// TIA Portal V20 export
VAR_GLOBAL   // PLC tag table "Unit1Em8"
   "BA060ZSIBK14.00" AT %I1052.0 : Bool;   // (HOME) HIPOT TAB CONTACTOR BACKWARD
   "BA060ZSIBK14.01" AT %I1052.1 : Bool;   // (HOME) HIPOT TAB CONTACTOR LEFT OPEN
   "BA060ZSIBK14.02" AT %I1052.2 : Bool;   // (HOME) HIPOT TAB CONTACTOR RIGHT OPEN
   "BA060ZSIBK14.03" AT %I1052.3 : Bool;   // SPARE
   "BA060ZSIBK14.04" AT %I1052.4 : Bool;   // SPARE
   "BA060ZSIBK14.05" AT %I1052.5 : Bool;   // (HOME) INSPECTION (HIPOT&THICKNESS) STAGE LIFT FRONT DOWN
   "BA060ZSIBK14.06" AT %I1052.6 : Bool;   // (HOME) INSPECTION (HIPOT&THICKNESS) STAGE LIFT REAR DOWN
   "BA060ZSIBK14.07" AT %I1052.7 : Bool;   // SPARE
   "BA060ZSIBK14.08" AT %I1053.0 : Bool;   // (WORK) HIPOT TAB CONTACTOR FORWARD
   "BA060ZSIBK14.09" AT %I1053.1 : Bool;   // (WORK) HIPOT TAB CONTACTOR LEFT CLOSE
   "BA060ZSIBK14.10" AT %I1053.2 : Bool;   // (WORK) HIPOT TAB CONTACTOR RIGHT CLOSE
   "BA060ZSIBK14.11" AT %I1053.3 : Bool;   // SPARE
   "BA060ZSIBK14.12" AT %I1053.4 : Bool;   // SPARE
   "BA060ZSIBK14.13" AT %I1053.5 : Bool;   // (WORK) INSPECTION (HIPOT&THICKNESS) STAGE LIFT FRONT UP
   "BA060ZSIBK14.14" AT %I1053.6 : Bool;   // (WORK) INSPECTION (HIPOT&THICKNESS) STAGE LIFT REAR UP
   "BA060ZSIBK14.15" AT %I1053.7 : Bool;   // SPARE
   "BA060ZSIBK15.02" AT %I1056.2 : Bool;   // HIPOT&THICKNESS STACK DETECT SENSOR
   "BA060ZSIBK15.03" AT %I1056.3 : Bool;   // HI-POT SAFETY PIN LOADING SENSOR
   "BA060ZSIBK15.04" AT %I1056.4 : Bool;   // SPARE
   "BA060ZSIBK15.05" AT %I1056.5 : Bool;   // SPARE
   "BA060ZSIBK15.06" AT %I1056.6 : Bool;   // SPARE
   "BA060ZSIBK15.07" AT %I1056.7 : Bool;   // SPARE
   "BA060ZSIBK15.09" AT %I1057.1 : Bool;   // SPARE
   "BA060ZSIBK15.10" AT %I1057.2 : Bool;   // SPARE
   "BA060ZSIBK15.11" AT %I1057.3 : Bool;   // SPARE
   "BA060ZSIBK15.12" AT %I1057.4 : Bool;   // SPARE
   "BA060ZSIBK15.13" AT %I1057.5 : Bool;   // SPARE
   "BA060ZSIBK15.14" AT %I1057.6 : Bool;   // SPARE
   "BA060ZSIBK15.15" AT %I1057.7 : Bool;   // SPARE
   "BA060AZSISP501.10" AT %I3001.0 : Bool;   // SPARE
   "BA060AZSISP501.11" AT %I3001.1 : Bool;   // SPARE
   "BA060AZSISP501.12" AT %I3001.2 : Bool;   // SPARE
   "BA060AZSISP501.13" AT %I3001.3 : Bool;   // SPARE
   "BA060AZSISP501.14" AT %I3001.4 : Bool;   // SPARE
   "BA060AZSISP501.15" AT %I3001.5 : Bool;   // SPARE
   "BA060AZSISP501.16" AT %I3001.6 : Bool;   // SPARE
   "BA060AZSISP501.17" AT %I3001.7 : Bool;   // SPARE
   "BA060ZSIPM08.00" AT %Q2028.0 : Bool;   // (WORK) HIPOT TAB CONTACTOR FORWARD
   "BA060ZSIPM08.01" AT %Q2028.1 : Bool;   // (HOME) HIPOT TAB CONTACTOR BACKWARD
   "BA060ZSIPM08.02" AT %Q2028.2 : Bool;   // (WORK) HIPOT TAB CONTACTOR LEFT CLOSE
   "BA060ZSIPM08.03" AT %Q2028.3 : Bool;   // (HOME) HIPOT TAB CONTACTOR LEFT OPEN
   "BA060ZSIPM08.04" AT %Q2028.4 : Bool;   // (WORK) HIPOT TAB CONTACTOR RIGHT CLOSE
   "BA060ZSIPM08.05" AT %Q2028.5 : Bool;   // (HOME) HIPOT TAB CONTACTOR RIGHT OPEN
   "BA060ZSIPM08.06" AT %Q2028.6 : Bool;   // SPARE
   "BA060ZSIPM08.07" AT %Q2028.7 : Bool;   // SPARE
   "BA060ZSIPM08.10" AT %Q2029.0 : Bool;   // SPARE
   "BA060ZSIPM08.11" AT %Q2029.1 : Bool;   // SPARE
   "BA060ZSIPM08.12" AT %Q2029.2 : Bool;   // (WORK) HIPOT & THICKNESS STAGE LIFT FRONT UP
   "BA060ZSIPM08.13" AT %Q2029.3 : Bool;   // (HOME) HIPOT & THICKNESS STAGE LIFT FRONT DOWN
   "BA060ZSIPM08.14" AT %Q2029.4 : Bool;   // (WORK) HIPOT & THICKNESS STAGE LIFT REAR DOWN
   "BA060ZSIPM08.15" AT %Q2029.5 : Bool;   // (HOME) HIPOT & THICKNESS STAGE LIFT REAR UP
   "BA060ZSIPM08.16" AT %Q2029.6 : Bool;   // SPARE
   "BA060ZSIPM08.17" AT %Q2029.7 : Bool;   // SPARE
   "BA060AZSISP504.10" AT %Q3001.0 : Bool;   // SPARE
   "BA060AZSISP504.11" AT %Q3001.1 : Bool;   // SPARE
   "BA060AZSISP504.12" AT %Q3001.2 : Bool;   // SPARE
   "BA060AZSISP504.13" AT %Q3001.3 : Bool;   // SPARE
   "BA060AZSISP504.14" AT %Q3001.4 : Bool;   // SPARE
   "BA060AZSISP504.15" AT %Q3001.5 : Bool;   // SPARE
   "BA060AZSISP504.16" AT %Q3001.6 : Bool;   // SPARE
   "BA060AZSISP504.17" AT %Q3001.7 : Bool;   // SPARE
END_VAR
VAR_GLOBAL CONSTANT   // user constants
   U1EM8_JOB01 : DInt := 1;   // ID for Job1
   U1EM8_JOB02 : DInt := 2;   // ID for Job2
   U1EM8_JOB03 : DInt := 3;   // ID for Job3
   U1EM8_JOB04 : DInt := 4;   // ID for Job4
   U1EM8_JOB05 : DInt := 5;   // ID for Job5
   U1EM8_JOB06 : DInt := 6;   // Starts with 1. E.g., the value means that axes exist.
   U1EM8_JOB07 : DInt := 7;
   U1EM8_JOB08 : DInt := 8;
   U1EM8_JOB09 : DInt := 9;
   U1EM8_JOB10 : DInt := 10;
   U1EM8_JOB11 : DInt := 11;
   U1EM8_JOB12 : DInt := 12;
   U1EM8_JOB13 : DInt := 13;
   U1EM8_JOB14 : DInt := 14;
   U1EM8_JOB15 : DInt := 15;
   U1EM8_JOB16 : DInt := 16;
   U1EM8_JOB17 : DInt := 17;
   U1EM8_JOB18 : DInt := 18;
   U1EM8_JOB19 : DInt := 19;
   U1EM8_JOB20 : DInt := 20;
   U1EM8_JOB21 : DInt := 21;
   U1EM8_JOB22 : DInt := 22;
   U1EM8_JOB23 : DInt := 23;
   U1EM8_JOB24 : DInt := 24;
   U1EM8_JOB25 : DInt := 25;
   U1EM8_JOB26 : DInt := 26;
   U1EM8_JOB27 : DInt := 27;
   U1EM8_JOB28 : DInt := 28;
   U1EM8_JOB29 : DInt := 29;
   U1EM8_JOB30 : DInt := 30;
   U1EM8_JOB31 : DInt := 31;
   U1EM8_JOB32 : DInt := 32;
   U1EM8_JOB33 : DInt := 33;
   U1EM8_JOB34 : DInt := 34;
   U1EM8_JOB35 : DInt := 35;
   U1EM8_JOB36 : DInt := 36;
   U1EM8_JOB37 : DInt := 37;
   U1EM8_JOB38 : DInt := 38;
   U1EM8_JOB39 : DInt := 39;
   U1EM8_JOB40 : DInt := 40;
   U1EM8_JOB41 : DInt := 41;
   U1EM8_JOB42 : DInt := 42;
   U1EM8_JOB43 : DInt := 43;
   U1EM8_JOB44 : DInt := 44;
   U1EM8_JOB45 : DInt := 45;
   U1EM8_JOB46 : DInt := 46;
   U1EM8_JOB47 : DInt := 47;
   U1EM8_JOB48 : DInt := 48;
   U1EM8_JOB49 : DInt := 49;
   U1EM8_JOB50 : DInt := 50;
   U1EM8_JOB51 : DInt := 51;
   U1EM8_JOB52 : DInt := 52;
   U1EM8_JOB53 : DInt := 53;
   U1EM8_JOB54 : DInt := 54;
   U1EM8_JOB55 : DInt := 55;
   U1EM8_JOB56 : DInt := 56;
   U1EM8_JOB57 : DInt := 57;
   U1EM8_JOB58 : DInt := 58;
   U1EM8_JOB59 : DInt := 59;
   U1EM8_JOB60 : DInt := 60;
   U1EM8_JOB61 : DInt := 61;
   U1EM8_JOB62 : DInt := 62;
   U1EM8_JOB63 : DInt := 63;
   U1EM8_JOB64 : DInt := 64;
   U1EM8_JOB65 : DInt := 65;
   U1EM8_JOB66 : DInt := 66;
   U1EM8_JOB67 : DInt := 67;
   U1EM8_JOB68 : DInt := 68;
   U1EM8_JOB69 : DInt := 69;
   U1EM8_JOB70 : DInt := 70;
   U1EM8_JOB71 : DInt := 71;
   U1EM8_JOB72 : DInt := 72;
   U1EM8_JOB73 : DInt := 73;
   U1EM8_JOB74 : DInt := 74;
   U1EM8_JOB75 : DInt := 75;
   U1EM8_JOB76 : DInt := 76;
   U1EM8_JOB77 : DInt := 77;
   U1EM8_JOB78 : DInt := 78;
   U1EM8_JOB79 : DInt := 79;
   U1EM8_JOB80 : DInt := 80;
   U1EM8_JOB81 : DInt := 81;
   U1EM8_JOB82 : DInt := 82;
   U1EM8_JOB83 : DInt := 83;
   U1EM8_JOB84 : DInt := 84;
   U1EM8_JOB85 : DInt := 85;
   U1EM8_JOB86 : DInt := 86;
   U1EM8_JOB87 : DInt := 87;
   U1EM8_JOB88 : DInt := 88;
   U1EM8_JOB89 : DInt := 89;
   U1EM8_JOB90 : DInt := 90;
   U1EM8_JOB91 : DInt := 91;
   U1EM8_JOB92 : DInt := 92;
   U1EM8_JOB93 : DInt := 93;
   U1EM8_JOB94 : DInt := 94;
   U1EM8_JOB95 : DInt := 95;
   U1EM8_JOB96 : DInt := 96;
   U1EM8_JOB97 : DInt := 97;
   U1EM8_JOB98 : DInt := 98;
   U1EM8_JOB99 : DInt := 99;
   U1EM8_SEQUENCE01 : Int := 1;
   U1EM8_SEQUENCE02 : Int := 2;
   U1EM8_SEQUENCE03 : Int := 3;
   U1EM8_SEQUENCE04 : Int := 4;
   U1EM8_SEQUENCE05 : Int := 5;
   U1EM8_SEQUENCE06 : Int := 6;
   U1EM8_SEQUENCE07 : Int := 7;
   U1EM8_SEQUENCE08 : Int := 8;
   U1EM8_SEQUENCE09 : Int := 9;
   U1EM8_SEQUENCE10 : Int := 10;
   U1EM8_SEQUENCE11 : Int := 11;
   U1EM8_SEQUENCE12 : Int := 12;
   U1EM8_SEQUENCE13 : Int := 13;
   U1EM8_SEQUENCE14 : Int := 14;
   U1EM8_SEQUENCE15 : Int := 15;
   U1EM8_SEQUENCE16 : Int := 16;
   U1EM8_SEQUENCE17 : Int := 17;
   U1EM8_SEQUENCE18 : Int := 18;
   U1EM8_SEQUENCE19 : Int := 19;
   U1EM8_SEQUENCE20 : Int := 20;
   U1EM8_SEQUENCE21 : Int := 21;
   U1EM8_SEQUENCE22 : Int := 22;
   U1EM8_SEQUENCE23 : Int := 23;
   U1EM8_SEQUENCE24 : Int := 24;
   U1EM8_SEQUENCE25 : Int := 25;
   U1EM8_SEQUENCE26 : Int := 26;
   U1EM8_SEQUENCE27 : Int := 27;
   U1EM8_SEQUENCE28 : Int := 28;
   U1EM8_SEQUENCE29 : Int := 29;
   U1EM8_SEQUENCE30 : Int := 30;
   U1EM8_SEQUENCE31 : Int := 31;
   U1EM8_SEQUENCE32 : Int := 32;
   U1EM8_SEQUENCE33 : Int := 33;
   U1EM8_SEQUENCE34 : Int := 34;
   U1EM8_SEQUENCE35 : Int := 35;
   U1EM8_SEQUENCE36 : Int := 36;
   U1EM8_SEQUENCE37 : Int := 37;
   U1EM8_SEQUENCE38 : Int := 38;
   U1EM8_SEQUENCE39 : Int := 39;
   U1EM8_SEQUENCE40 : Int := 40;
   U1EM8_SEQUENCE41 : Int := 41;
   U1EM8_SEQUENCE42 : Int := 42;
   U1EM8_SEQUENCE43 : Int := 43;
   U1EM8_SEQUENCE44 : Int := 44;
   U1EM8_SEQUENCE45 : Int := 45;
   U1EM8_SEQUENCE46 : Int := 46;
   U1EM8_SEQUENCE47 : Int := 47;
   U1EM8_SEQUENCE48 : Int := 48;
   U1EM8_SEQUENCE49 : Int := 49;
   U1EM8_SEQUENCE50 : Int := 50;
   U1EM8_SEQUENCE51 : Int := 51;
   U1EM8_SEQUENCE52 : Int := 52;
   U1EM8_SEQUENCE53 : Int := 53;
   U1EM8_SEQUENCE54 : Int := 54;
   U1EM8_SEQUENCE55 : Int := 55;
   U1EM8_SEQUENCE56 : Int := 56;
   U1EM8_SEQUENCE57 : Int := 57;
   U1EM8_SEQUENCE58 : Int := 58;
   U1EM8_SEQUENCE59 : Int := 59;
   U1EM8_SEQUENCE60 : Int := 60;
   U1EM8_SEQUENCE61 : Int := 61;
   U1EM8_SEQUENCE62 : Int := 62;
   U1EM8_SEQUENCE63 : Int := 63;
   U1EM8_SEQUENCE64 : Int := 64;
   U1EM8_SEQUENCE65 : Int := 65;
   U1EM8_SEQUENCE66 : Int := 66;
   U1EM8_SEQUENCE67 : Int := 67;
   U1EM8_SEQUENCE68 : Int := 68;
   U1EM8_SEQUENCE69 : Int := 69;
   U1EM8_SEQUENCE70 : Int := 70;
   U1EM8_SEQUENCE71 : Int := 71;
   U1EM8_SEQUENCE72 : Int := 72;
   U1EM8_SEQUENCE73 : Int := 73;
   U1EM8_SEQUENCE74 : Int := 74;
   U1EM8_SEQUENCE75 : Int := 75;
   U1EM8_SEQUENCE76 : Int := 76;
   U1EM8_SEQUENCE77 : Int := 77;
   U1EM8_SEQUENCE78 : Int := 78;
   U1EM8_SEQUENCE79 : Int := 79;
   U1EM8_SEQUENCE80 : Int := 80;
   U1EM8_SEQUENCE81 : Int := 81;
   U1EM8_SEQUENCE82 : Int := 82;
   U1EM8_SEQUENCE83 : Int := 83;
   U1EM8_SEQUENCE84 : Int := 84;
   U1EM8_SEQUENCE85 : Int := 85;
   U1EM8_SEQUENCE86 : Int := 86;
   U1EM8_SEQUENCE87 : Int := 87;
   U1EM8_SEQUENCE88 : Int := 88;
   U1EM8_SEQUENCE89 : Int := 89;
   U1EM8_SEQUENCE90 : Int := 90;
   U1EM8_SEQUENCE91 : Int := 91;
   U1EM8_SEQUENCE92 : Int := 92;
   U1EM8_SEQUENCE93 : Int := 93;
   U1EM8_SEQUENCE94 : Int := 94;
   U1EM8_SEQUENCE95 : Int := 95;
   U1EM8_SEQUENCE96 : Int := 96;
   U1EM8_SEQUENCE97 : Int := 97;
   U1EM8_SEQUENCE98 : Int := 98;
   U1EM8_SEQUENCE99 : Int := 99;
   U1EM8_NO_OF_SEQUENCE : USInt := 0;
   U1EM8_NO_OF_AXES : USInt := 1;
END_VAR
